FUNCTION_BLOCK TLCtrlWait (* a simple FB Function Block Type *)
  (* Standard: 61499-1; Type: Simple FB; Description: Template for a Simple FB *)
  (* Version 0.2, 2020-05-24, JHC, Holobloc Inc, Added ECC documentation. *)
  (* Version 0.1, 2020-05-19, JHC, Holobloc Inc, Changed name from SimpleFB back to Simple. *)
  (* Version 0.0, 2020-05-05, JHC, Holobloc Inc *)
  PACKAGE fb.rt.myfb;
  IMPORT fb.datatype.*;
  IMPORT fb.rt.*;
  (* Compiler Java AdoptOpenJDK JDK 1.8.0_222 *)
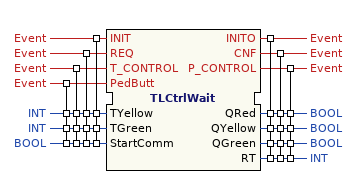
  EVENT_INPUT
    INIT WITH TYellow, TGreen, StartComm; (* Service Initialization *)
    REQ WITH TYellow, TGreen, StartComm; (* Service Request *)
    T_CONTROL WITH TYellow, TGreen, StartComm;
    PedButt WITH TYellow, TGreen, StartComm;
  END_EVENT
  EVENT_OUTPUT
    INITO WITH QRed, QYellow, QGreen, RT; (* Initialization Confirm *)
    CNF WITH QRed, QYellow, QGreen, RT; (* Confirmation of Requested Service *)
    P_CONTROL WITH QRed, QYellow, QGreen, RT;
  END_EVENT
  VAR_INPUT
    TYellow : INT; (* Event Input Qualifier *)
    TGreen : INT; (* Input Variable *)
    StartComm : BOOL;
  END_VAR
  VAR_OUTPUT
    QRed : BOOL; (* Event Output Qualifier *)
    QYellow : BOOL; (* Service Status *)
    QGreen : BOOL; (* Output variable *)
    RT : INT;
  END_VAR
  VAR
    CountVar : INT;
    Step : INT;
    pom : BOOL;
  END_VAR
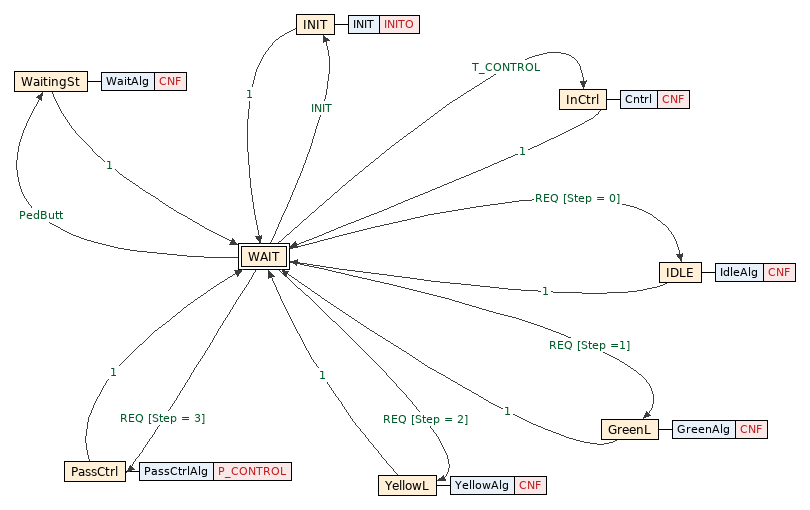
  EC_STATES
    WAIT;
    IDLE : IdleAlg -> CNF;
    INIT : INIT -> INITO;
    InCtrl : Cntrl -> CNF;
    GreenL : GreenAlg -> CNF;
    YellowL : YellowAlg -> CNF;
    PassCtrl : PassCtrlAlg -> P_CONTROL;
    WaitingSt : WaitAlg -> CNF;
  END_STATES
  EC_TRANSITIONS
    WAIT TO IDLE := REQ [Step = 0];
    WAIT TO INIT := INIT;
    INIT TO WAIT := 1;
    IDLE TO WAIT := 1;
    WAIT TO InCtrl := T_CONTROL;
    InCtrl TO WAIT := 1;
    WAIT TO GreenL := REQ [Step =1];
    GreenL TO WAIT := 1;
    WAIT TO YellowL := REQ [Step = 2];
    YellowL TO WAIT := 1;
    WAIT TO PassCtrl := REQ [Step = 3];
    PassCtrl TO WAIT := 1;
    WAIT TO WaitingSt := PedButt;
    WaitingSt TO WAIT := 1;
  END_TRANSITIONS
  ALGORITHM INIT IN ST: (* Initialization Algorithm *)
IF StartComm = TRUE THEN
	Step := 1;
	CountVar := 0;
ELSE
	Step := 0;
	CountVar := 0;
END_IF
  END_ALGORITHM
  ALGORITHM IdleAlg IN ST: (* Normally Executed Algorithm *)
QRed := TRUE;
QYellow := FALSE;
QGreen := FALSE;

RT := 0;
  END_ALGORITHM
  ALGORITHM GreenAlg IN ST:
CountVar := CountVar + 1;

QRed := FALSE;
QYellow := FALSE;
QGreen := TRUE;

RT := TGreen - CountVar;

IF RT <= 0 OR (pom AND CountVar >=4) THEN
	CountVar := 0;
	pom := FALSE;
	Step := 2;
END_IF
  END_ALGORITHM
  ALGORITHM Cntrl IN ST:
Step := 1;
  END_ALGORITHM
  ALGORITHM YellowAlg IN ST:
CountVar := CountVar + 1;

QRed := FALSE;
QYellow := TRUE;
QGreen := FALSE;

RT := TYellow - CountVar;

IF RT <= 0 THEN
	CountVar := 0;
	Step := 3;
END_IF
  END_ALGORITHM
  ALGORITHM PassCtrlAlg IN ST:
CountVar := 0;
Step := 0;
  END_ALGORITHM
  ALGORITHM WaitAlg IN ST:
pom := TRUE;
  END_ALGORITHM
END_FUNCTION_BLOCK
